// Mitsubishi GX Works2 project: 응용1   PLC: Q02/Q02H

PROGRAM MAIN
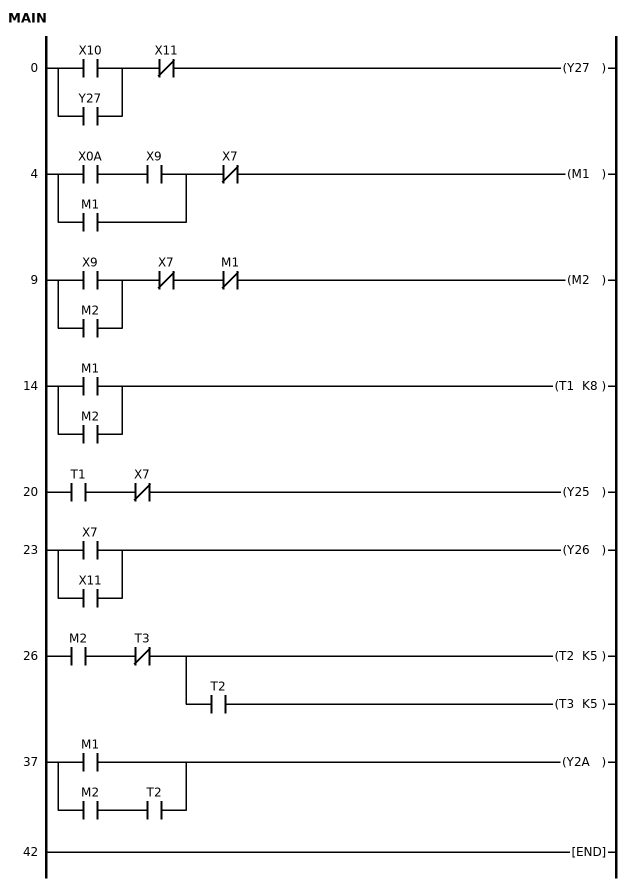
0     LD      X10
      OR      Y27
      ANI     X11
      OUT     Y27
4     LD      X0A
      AND     X9
      OR      M1
      ANI     X7
      OUT     M1
9     LD      X9
      OR      M2
      ANI     X7
      ANI     M1
      OUT     M2
14    LD      M1
      OR      M2
      OUT     T1 K8
20    LD      T1
      ANI     X7
      OUT     Y25
23    LD      X7
      OR      X11
      OUT     Y26
26    LD      M2
      ANI     T3
      OUT     T2 K5
      AND     T2
      OUT     T3 K5
37    LD      M1
      LD      M2
      AND     T2
      ORB
      OUT     Y2A
42    END
END_PROGRAM
